TYPE Homing_CoE_Ctrl_Paramters_typ :
STRUCT
	HomingMethod  : SINT; 
	HomingSWSpeed : UDINT;
	HomingTrSpeed : UDINT; 
	HomingAcc     : UDINT;
	HomingOffset  : DINT;
 
END_STRUCT
END_TYPE

(* stored: Version 1.1.0.1, ProductVersion 3.1.4024.3
   DUT Homing_CoE_Ctrl_Paramters_typ: Id {baed6811-c21c-0f67-1f54-7e24a06daf8f} *)
